{attribute 'linkalways'} 
{attribute 'no_explicit_call' := 'This FB is a CLASS and must be accessed using methods or properties'}
{attribute 'enable_dynamic_creation'}
FUNCTION_BLOCK _ITcVnBidirectionalIterator EXTENDS InterfaceDatatypeBase IMPLEMENTS I_InterfaceDatatype_ITcVnBidirectionalIterator
VAR
	localData : ITcVnBidirectionalIterator;
	activeData : REFERENCE TO ITcVnBidirectionalIterator REF= localData;
END_VAR

PROPERTY PUBLIC Address : PVOID
GET
Address := ADR(activeData);
END_GET
END_PROPERTY

METHOD PUBLIC ClearReference
VAR_INPUT
END_VAR
activeData REF= localData;
END_METHOD

METHOD PUBLIC Clone : I_Datatype
VAR
    pClone : POINTER TO _ITcVnBidirectionalIterator;
END_VAR
pClone := __NEW(_ITcVnBidirectionalIterator);
Clone := pClone^;
END_METHOD

METHOD FB_exit : BOOL
VAR_INPUT
	bInCopyCode : BOOL; // if TRUE, the exit method is called for exiting an instance that is copied afterwards (online change).
END_VAR
IF bInCopyCode THEN
	RETURN;
END_IF

TryTcReleaseLocal();
END_METHOD

PROPERTY PUBLIC Identifier : T_MAXSTRING
GET
Identifier := 'ITcVnBidirectionalIterator';
END_GET
END_PROPERTY

PROPERTY PUBLIC IsValid : BOOL
GET
IsValid := activeData <> 0;
END_GET
END_PROPERTY

METHOD PUBLIC MakeReferenceTo
VAR_INPUT
	ReferenceTarget : REFERENCE TO ITcVnBidirectionalIterator;
END_VAR
activeData REF= ReferenceTarget;
END_METHOD

METHOD PUBLIC SerializeWith
VAR_INPUT
	Serializer : I_Serializer;
END_VAR
Serializer.AddNull();
END_METHOD

PROPERTY PUBLIC Size : UDINT
GET
Size := SIZEOF(activeData);
END_GET
END_PROPERTY

METHOD PUBLIC TryCheckIfBegin : BOOL
VAR_INPUT
	Result : REFERENCE TO BOOL;
END_VAR
Result := FALSE;

IF NOT IsValid THEN
	RETURN;
END_IF

IF activeData.CheckIfBegin() = S_OK THEN
    Result := TRUE;
END_IF

TryCheckIfBegin := TRUE;
END_METHOD

METHOD PUBLIC TryCheckIfEnd : BOOL
VAR_INPUT
	Result : REFERENCE TO BOOL;
END_VAR
Result := FALSE;

IF NOT IsValid THEN
	RETURN;
END_IF

IF activeData.CheckIfEnd() = S_OK THEN
    Result := TRUE;
END_IF

TryCheckIfEnd := TRUE;
END_METHOD

METHOD PUBLIC TryCopyContentFrom : BOOL
VAR_INPUT
	Source : I_InterfaceDatatype;
END_VAR
// currently un-copyable
END_METHOD

METHOD TryDeserializeFrom : BOOL
VAR_INPUT
	Deserializer : I_Deserializer;
	Feedback : I_DeserializerFeedback;
END_VAR
VAR
END_VAR
// not implemented.
END_METHOD

METHOD PUBLIC TryGetValueSize : BOOL
VAR_INPUT
	Destination : REFERENCE TO ULINT;
END_VAR
IF NOT IsValid THEN
	RETURN;
END_IF

TryGetValueSize := SUCCEEDED(activeData.GetValueSize(Destination));
END_METHOD

METHOD PUBLIC TryGetValueTypeGuid : BOOL
VAR_INPUT
	Destination : REFERENCE TO GUID;
END_VAR
IF NOT IsValid THEN
	RETURN;
END_IF

TryGetValueTypeGuid := SUCCEEDED(activeData.GetValueTypeGuid(Destination));
END_METHOD

METHOD TryMakeReferenceTo : BOOL
VAR_INPUT
	Target : I_Datatype;
END_VAR
VAR
	pTargetData : POINTER TO ITcVnBidirectionalIterator;
END_VAR
IF NOT IsEquivalentTo(Target) THEN
	RETURN;
END_IF

pTargetData := Target.Address;
activeData REF= pTargetData^;
TryMakeReferenceTo := TRUE;
END_METHOD

METHOD PUBLIC TryTcAddRef : BOOL
VAR_INPUT
END_VAR
IF activeData = 0 THEN
	RETURN;
END_IF

IF activeData.TcAddRef() = 0 THEN
	activeData := 0;
END_IF

TryTcAddRef := TRUE;
END_METHOD

METHOD PUBLIC TryTcRelease : BOOL
VAR_INPUT
END_VAR
IF activeData = 0 THEN
	RETURN;
END_IF

IF activeData.TcRelease() = 0 THEN
	activeData := 0;
END_IF

TryTcRelease := TRUE;
END_METHOD

METHOD PUBLIC TryTcReleaseLocal : BOOL
VAR_INPUT
END_VAR
IF localData = 0 THEN
	RETURN;
END_IF

IF localData.TcRelease() = 0 THEN
	localData := 0;
END_IF

TryTcReleaseLocal := TRUE;
END_METHOD

PROPERTY PUBLIC Value : REFERENCE TO ITcVnBidirectionalIterator
GET
Value REF= activeData;
END_GET
END_PROPERTY

END_FUNCTION_BLOCK

(* stored: Version 1.1.0.1, ProductVersion 3.1.4026.13
   POU _ITcVnBidirectionalIterator: Id {34fa7641-846d-0f2d-14a7-eb5fd9e7b60b}, SpecialFunc None
   Folder Core: Id {3c3e4c0d-3d4c-0c92-02bb-1d1f91afbf8f}
   Folder Customize: Id {f5b39792-d60f-08cb-18aa-d640e9b22c64}
   Folder Destructor: Id {ffe022f9-f833-04d5-361a-d03789118cd9}
   Folder Private: Id {0a3fc2d3-7068-0e0d-0d86-53f4e3fbdb7c}
   Property Address: Id {0bc03280-c56c-0cc7-1afc-2edfa5c4065c}
   Get Get: Id {588d7efa-e9d0-0138-1bca-40d831b78127}
   Method ClearReference: Id {1be49da6-880f-0325-3534-79fcc06f3725}
   Method Clone: Id {63eba12a-1568-018f-0f62-bd94ca985c71}
   Method FB_exit: Id {4c61ab2f-4ec8-0c8a-2567-2ae40a44cb13}
   Property Identifier: Id {c6491e99-8fcd-011a-0641-7f8906efa1f2}
   Get Get: Id {daad6b6c-7d60-08a7-1cfd-06fba8172505}
   Property IsValid: Id {1d127891-191b-0c31-1c87-e19954f1bc2c}
   Get Get: Id {9c547f0c-b6db-0cad-1245-7c4fefbbfe7c}
   Method MakeReferenceTo: Id {7c4005a3-37df-0f6d-0e4f-0d5e798eaefa}
   Method SerializeWith: Id {8e9329da-eab9-00d9-21b8-cda7ba62f2b8}
   Property Size: Id {200e36e7-6134-0a1c-288d-b8c8b395f4cd}
   Get Get: Id {073c4832-a9b3-0b8a-27e4-9ca0b81371bf}
   Method TryCheckIfBegin: Id {919bc0d9-ee18-0c51-1821-35727836149d}
   Method TryCheckIfEnd: Id {474b55af-afd8-084a-0c9c-49eb2d87ce2d}
   Method TryCopyContentFrom: Id {51e2e2b3-4d91-0427-3957-0e352c8c56e4}
   Method TryDeserializeFrom: Id {80135932-bf49-0807-173d-d8d33f54eaef}
   Method TryGetValueSize: Id {3f8b3462-c21b-0d4e-24bd-7d84b6729db6}
   Method TryGetValueTypeGuid: Id {2c251413-61ea-097d-0d3e-3f869278b99d}
   Method TryMakeReferenceTo: Id {d87be40b-a47b-026b-2474-7e298495e425}
   Method TryTcAddRef: Id {4cbee62f-07bb-0711-334d-d7a0ff3c2367}
   Method TryTcRelease: Id {4e7234b9-453b-034a-3b58-a96e9766d8cf}
   Method TryTcReleaseLocal: Id {3eb3c7d9-e6bf-02bd-31c4-dba785773f57}
   Property Value: Id {09fb64ad-20a5-0b4b-2618-efca8aebee96}
   Get Get: Id {b42e398f-e4be-05a2-299f-321a712d042d} *)
